PROGRAM testProg
VAR
END_VAR

END_PROGRAM

(* stored: Version 1.1.0.1, ProductVersion 3.1.4024.5
   POU testProg: Id {6b742e2c-3720-4a26-aa80-15486c69d838}, SpecialFunc None *)
